Fanuc TP program (LS listing): BLANK.LS

/PROG  ABC

/ATTR

OWNER		= MNEDITOR;

COMMENT		= "";

PROG_SIZE	= 0;

CREATE		= DATE 120-11-14  TIME 14:26:01;

MODIFIED	= DATE 121-03-07  TIME 08:28:09;

FILE_NAME	= ;

VERSION		= 0;

LINE_COUNT	= 0;

MEMORY_SIZE	= 314;

PROTECT		= READ_WRITE;

TCD:  STACK_SIZE	= 0,

      TASK_PRIORITY	= 50,

      TIME_SLICE	= 0,

      BUSY_LAMP_OFF	= 0,

      ABORT_REQUEST	= 0,

      PAUSE_REQUEST	= 0;

DEFAULT_GROUP	= 1,*,*,*,*;

CONTROL_CODE	= 00000000 00000000;

/MN

/POS

/END
